// TIA Portal V17 export
// export: Created 2025-06-26T06:49:21.0323822Z, ExportSetting WithDefaults, DisplayName Totally Integrated Automation Portal, DisplayVersion V17 Update 8, DisplayName TIA Portal Openness, DisplayVersion V17 Update 8, DisplayName TIA Portal Version Control Interface, DisplayVersion V17, DisplayName STEP 7 Professional, DisplayVersion V17 Update 8, DisplayName STEP 7 Safety, DisplayVersion V17 Update 6, DisplayName WinCC Advanced, DisplayVersion V17 Update 8
DATA_BLOCK "Cloud_DB"   // DB15
VERSION : 0.1
// stored: AutoNumber true, DBAccessibleFromOPCUA true, InstanceOfName Cloud, InstanceOfType FB
"Cloud"
   // VAR
   //    CurrentTime { ExternalWritable := 'False'} : DTL;
   //    SetTime : DTL;
   //    Update : Bool;
   // END_VAR
BEGIN
END_DATA_BLOCK
